PROGRAM MAIN
VAR

inc1 : DINT := 0;

	
END_VAR

GVL.mOutTrain := GVL.mInTrain;

//0 to 37 map to blocks 1-38
//38 to 43 map to 72-76,yard
//Lights Logic
FOR inc1 := 0 TO 43 DO
	//Sets Red Lights
	IF GVL.mInOccupancies[inc1] = 1
	THEN
		GVL.mOutLeftLights[inc1] := 0;
		GVL.mOutRightLights[inc1] := 0;
	//Sets green lights
	ELSE
		GVL.mOutLeftLights[inc1] := 2;
		GVL.mOutRightLights[inc1] := 2;
	END_IF
END_FOR

FOR inc1 := 1 TO 43 DO
	//Sets Yellow Lights
	IF GVL.mInOccupancies[inc1-1] = 1 AND GVL.mInOccupancies[inc1] <> 1
	THEN
		GVL.mOutRightLights[inc1] := 1;
	END_IF
	IF GVL.mInOccupancies[inc1+1] = 1 AND GVL.mInOccupancies[inc1] <> 1
	THEN
	GVL.mOutLeftLights[inc1] := 1;
	END_IF
END_FOR

//0 to 37 map to blocks 1-38
//39 to 43 map to blocks 72-76,yard
//Passes occupancy, authority, maintenance, and speeds from input to output.
FOR inc1 := 0 TO 43 DO
	
	GVL.mOutOccupancies[inc1] := GVL.mInOccupancies[inc1];
	GVL.mOutAuthorities[inc1] := GVL.mInAuthorities[inc1];
	GVL.mOutMaintenance[inc1] := GVL.mInMaintenance[inc1];
	IF GVL.mInSpeeds[inc1] < GVL.mSpeedLimits[inc1] AND GVL.mInSpeeds[inc1] <> 0
	THEN
		GVL.mOutSpeeds[inc1] := GVL.mInSpeeds[inc1];
	ELSE
		GVL.mOutSpeeds[inc1] := GVL.mSpeedLimits[inc1];
	END_IF
	
END_FOR

FOR inc1 := 0 TO 43 DO

	GVL.mOutRoute[inc1] := GVL.mInRoute[inc1];
	
END_FOR

inc1 := 0;

//This starts the main track logic section

//0 to 37 map to blocks 1-38
//39 to 43 map to 72-76,yard
//Switch Logic
IF GVL.mInMaintenance[8] = 1 
THEN
	IF GVL.mInSwitch[8] = 1
	THEN
		IF GVL.mOutSwitch[8] = 9
			THEN
			GVL.mOutSwitch[8] := 76;
			GVL.mInSwitch[8] := 0;
		ELSE
			GVL.mOutSwitch[8] := 9;
			GVL.mInSwitch[8] := 0;
		END_IF
	END_IF
ELSE
    IF GVL.mInOccupancies[43] = 1 
	THEN
    	GVL.mOutSwitch[8] := 76;
    ELSE
		GVL.mOutSwitch[8] := 9;
	END_IF
END_IF

//0 to 37 map to blocks 1-38
//39 to 43 map to 72-76,yard
IF GVL.mInMaintenance[15] = 1 
THEN
    IF GVL.mInSwitch[15] = 1
	THEN
		IF GVL.mOutSwitch[15] = 0
			THEN
			GVL.mOutSwitch[15] := 16;
			GVL.mInSwitch[15] := 0;
		ELSE
			GVL.mOutSwitch[15] := 0;
			GVL.mInSwitch[15] := 0;
		END_IF
	END_IF
ELSE
    IF GVL.mInOccupancies[14] = 1 
	THEN
	    GVL.mOutSwitch[15] := 14;
    ELSE
        GVL.mOutSwitch[15] := 0;
    END_IF
END_IF

//0 to 37 map to blocks 1-38
//39 to 43 map to 72-76,yard
IF GVL.mInMaintenance[26] = 1 
THEN
    IF GVL.mInSwitch[26] = 1
	THEN
		IF GVL.mOutSwitch[26] = 75
			THEN
			GVL.mOutSwitch[26] := 27;
			GVL.mInSwitch[26] := 0;
		ELSE
			GVL.mOutSwitch[26] := 75;
			GVL.mInSwitch[26] := 0;
		END_IF
	END_IF
ELSE
    IF GVL.mInOccupancies[42] = 1 
	THEN
	    GVL.mOutSwitch[26] := 75;
    ELSE
        GVL.mOutSwitch[26] := 27;
    END_IF
END_IF

//0 to 37 map to blocks 1-38
//39 to 43 map to 72-76,yard
IF GVL.mInMaintenance[32] = 1 
THEN
  IF GVL.mInSwitch[32] = 1
	THEN
		IF GVL.mOutSwitch[32] = 31
			THEN
			GVL.mOutSwitch[32] := 71;
			GVL.mInSwitch[32] := 0;
		ELSE
			GVL.mOutSwitch[32] := 31;
			GVL.mInSwitch[32] := 0;
		END_IF
	END_IF
ELSE
    IF GVL.mInOccupancies[31] = 1 
	THEN
	    GVL.mOutSwitch[32] := 31;
    ELSE
        GVL.mOutSwitch[32] := 71;
    END_IF
END_IF

END_PROGRAM

(* stored: Version 1.1.0.1, ProductVersion 3.1.4024.11
   POU MAIN: Id {fa45f2f2-925a-467e-8b80-1fe2692585de}, SpecialFunc None *)
